PROGRAM ProgramTask2
VAR
	nRead : udint;
END_VAR

ProgramTask1.ipSpscBuff.Get(ADR(nRead),SIZEOF(nRead));

END_PROGRAM

(* stored: Version 1.1.0.1
   POU ProgramTask2: Id {1bd251a5-443a-4986-869e-8395af033291}, SpecialFunc None *)
